ABB RAPID module: Wobj_FRAME_BufferC.mod

MODULE Wobj_FRAME_BufferC
	! Points are read in order of declaration.
  ! Please do not change the order of points!

  LOCAL PERS robtarget pWobj_U_PointX1:=[[1633.529,-1257.445,116.3468],[0.0103661855682731,-0.306948602199554,0.951647579669952,0.00647602137178183],[-1,0,-1,0],[9E+09,9E+09,9E+09,9E+09,9E+09,9E+09]];
	LOCAL PERS robtarget pWobj_U_PointX2:=[[-1961.429,-1284.259,120.119],[0.0119650475680828,-0.87871652841568,0.477187633514404,-0.0024547167122364],[-2,-1,1,0],[9E+09,9E+09,9E+09,9E+09,9E+09,9E+09]];
	LOCAL PERS robtarget pWobj_U_PointY1:=[[1639.556,-2455.425,116.8528],[0.0103659750893712,-0.30694243311882,0.95164954662323,0.00647744350135326],[-1,0,-2,0],[9E+09,9E+09,9E+09,9E+09,9E+09,9E+09]];

ENDMODULE
